{attribute addProperty BoxType "EK1100-0000-0018"}
{attribute addProperty Id "Beckhoff_EL37xxEK1122Beckhoff_EL37xxEK1122_36723BB4162A_0001_EL3702_0000_0002EL3702_C61743E644856A_0002_EL3702_0000_0003EL3702_C61743E644856A_0003_EL3702_0015_0003EL3702_C61743E644856A_0004_EL3742_0000_0001EL3742_FE433AD517622A_0005_EL3742_0000_0002EL3742_C61743E644856A_0006_EL3742_0000_0003EL3742_C61743E644856A_0007_EL3751_0000_0020EL3751_3EC4001E28836A_0008_EL3751_0000_0021EL3751_3EC4001E28836A_0009_EL3751_0000_0022EL3751_3EC4001E28836A_0010_EL3751_0000_0023EL3751_3EC4001E28836A_0011_EL3751_0004_0022EL3751_3EC4001E28836A_0012_EL3751_0004_0023EL3751_3EC4001E28836A_0013_EL3751_0020_0020EL3751_3EC4001E28836A_0014_EL3751_0020_0021EL3751_3EC4001E28836A_0015_EL3751_0020_0022EL3751_3EC4001E28836A_0016_EL3751_0020_0023EL3751_3EC4001E28836A_0017_EL3751_0024_0022EL3751_3EC4001E28836A_0018_EL3751_0024_0023EL3751_3EC4001E28836A_0019_EL3773_0000_0016EL3773_D84CC94E1296162A_0020_EL3773_0000_0017EL3773_2453D1BA1296162A_0021_EL3773_0000_0018EL3773_0A81905D1296162A_0022_EL3773_0000_0019EL3773_8352C0071296162A_0023_EL3773_0000_0020EL3773_8352C0071296162A_0024_EL3773_0000_0021EL3773_8352C0071296162A_0025_EL3783_0000_0018EL3783_F9BCA3512296287"}
{attribute addProperty CRC "4017479005"}
{attribute addProperty SizeInBites "15960"}
{attribute addProperty SizeInBytes "1995"}
TYPE Beckhoff_EL37xx_EF75DD5D EXTENDS EK1100_179A0949 :
STRUCT
	{attribute addProperty Name "Beckhoff_EL37xxEK1122"}
	Beckhoff_EL37xxEK1122 : Beckhoff_EL37xxEK1122_36723BB4;
	{attribute addProperty Name "A_0001_EL3702_0000_0002"}
	A_0001_EL3702_0000_0002 : EL3702_C61743E6;
	{attribute addProperty Name "A_0002_EL3702_0000_0003"}
	A_0002_EL3702_0000_0003 : EL3702_C61743E6;
	{attribute addProperty Name "A_0003_EL3702_0015_0003"}
	A_0003_EL3702_0015_0003 : EL3702_C61743E6;
	{attribute addProperty Name "A_0004_EL3742_0000_0001"}
	A_0004_EL3742_0000_0001 : EL3742_FE433AD5;
	{attribute addProperty Name "A_0005_EL3742_0000_0002"}
	A_0005_EL3742_0000_0002 : EL3742_C61743E6;
	{attribute addProperty Name "A_0006_EL3742_0000_0003"}
	A_0006_EL3742_0000_0003 : EL3742_C61743E6;
	{attribute addProperty Name "A_0007_EL3751_0000_0020"}
	A_0007_EL3751_0000_0020 : EL3751_3EC4001E;
	{attribute addProperty Name "A_0008_EL3751_0000_0021"}
	A_0008_EL3751_0000_0021 : EL3751_3EC4001E;
	{attribute addProperty Name "A_0009_EL3751_0000_0022"}
	A_0009_EL3751_0000_0022 : EL3751_3EC4001E;
	{attribute addProperty Name "A_0010_EL3751_0000_0023"}
	A_0010_EL3751_0000_0023 : EL3751_3EC4001E;
	{attribute addProperty Name "A_0011_EL3751_0004_0022"}
	A_0011_EL3751_0004_0022 : EL3751_3EC4001E;
	{attribute addProperty Name "A_0012_EL3751_0004_0023"}
	A_0012_EL3751_0004_0023 : EL3751_3EC4001E;
	{attribute addProperty Name "A_0013_EL3751_0020_0020"}
	A_0013_EL3751_0020_0020 : EL3751_3EC4001E;
	{attribute addProperty Name "A_0014_EL3751_0020_0021"}
	A_0014_EL3751_0020_0021 : EL3751_3EC4001E;
	{attribute addProperty Name "A_0015_EL3751_0020_0022"}
	A_0015_EL3751_0020_0022 : EL3751_3EC4001E;
	{attribute addProperty Name "A_0016_EL3751_0020_0023"}
	A_0016_EL3751_0020_0023 : EL3751_3EC4001E;
	{attribute addProperty Name "A_0017_EL3751_0024_0022"}
	A_0017_EL3751_0024_0022 : EL3751_3EC4001E;
	{attribute addProperty Name "A_0018_EL3751_0024_0023"}
	A_0018_EL3751_0024_0023 : EL3751_3EC4001E;
	{attribute addProperty Name "A_0019_EL3773_0000_0016"}
	A_0019_EL3773_0000_0016 : EL3773_D84CC94E;
	{attribute addProperty Name "A_0020_EL3773_0000_0017"}
	A_0020_EL3773_0000_0017 : EL3773_2453D1BA;
	{attribute addProperty Name "A_0021_EL3773_0000_0018"}
	A_0021_EL3773_0000_0018 : EL3773_0A81905D;
	{attribute addProperty Name "A_0022_EL3773_0000_0019"}
	A_0022_EL3773_0000_0019 : EL3773_8352C007;
	{attribute addProperty Name "A_0023_EL3773_0000_0020"}
	A_0023_EL3773_0000_0020 : EL3773_8352C007;
	{attribute addProperty Name "A_0024_EL3773_0000_0021"}
	A_0024_EL3773_0000_0021 : EL3773_8352C007;
	{attribute addProperty Name "A_0025_EL3783_0000_0018"}
	A_0025_EL3783_0000_0018 : EL3783_F9BCA351;
END_STRUCT
END_TYPE

(* stored: Version 1.2.0.0, ProductVersion 3.1.4024.9
   DUT Beckhoff_EL37xx_EF75DD5D: Id {1ed9b2d6-4828-4734-ae86-6bf1c26416bf} *)
